FUNCTION_BLOCK FB_FeedForward
VAR_INPUT
	fXDotRef 	: LREAL; // Motion Referance
	fQMaxUp 	: LREAL; // Needs to be positive (22)
	fQMaxDown 	: LREAL; // Needs to be positive (15)
	fDeadUp		: LREAL; // Needs to be positive (0.155)
	fDeadDown 	: LREAL; // Needs to be positive (0.18)
	fPs 		: LREAL;
	fPa			: LREAL;
	fPb			: LREAL;
	fKFF 		: LREAL; // Coefficient of FeedForward
END_VAR
VAR_OUTPUT
	fUFF : LREAL;
END_VAR
VAR
	fUTemp : LREAL;
	fUMax : LREAL := 0.9;
	fQRef : LREAL;
	fAp : LREAL := 33.1 / 10000.0;
	fAa : LREAL := 23.56 / 10000.0;
	
	fK02Up : LREAL := 0.78; //0.78;
	fK04Up : LREAL := 2.29; //2.3;
	fK06Up : LREAL := 3.42;// 3.27;
	fK07Up : LREAL := 4.59; //4.54;
	fK08Up : LREAL := 5.09; //4.94;
	fK1Up : LREAL := 5.71; //5.68;
	
	fK02Down : LREAL := -0.75; //-0.75; 
	fK04Down : LREAL := -2.17; //-2.21; //-1.37;
	fK06Down : LREAL := -3.39; //-3.45; 
	fK07Down : LREAL := -3.99; //-3.96; //-2.45;
	fK08Down : LREAL := -4.55; //-4.61; 
	fK1Down : LREAL := -4.84; //-4.67; //-2.88;
	
	fDeltaP : LREAL;
	fKRef : LREAL; 
	
END_VAR



IF fXDotRef >= 0.0 THEN // Upwards
	
	fQRef := fAp * fXDotRef * 60000;
	fDeltaP := fPs - fPa;
	IF fDeltaP < 100 THEN
		fDeltaP := 100;
	ELSE
		fDeltaP := fDeltaP;
	END_IF
	fKRef := fQRef / SQRT(fDeltaP);
	
	IF fKRef < 0.0 THEN
		fUTemp := 0.0;
	ELSIF fKRef < fK02Up THEN
		fUTemp := -fKRef/fK02Up * (0.2 - fDeadUp);
	ELSIF fKRef < fK04Up THEN
		fUTemp := -(0.2 - fDeadUp) -(fKRef - fK02Up) / (fK04Up - fK02Up) * (0.4-fDeadUp-0.2);
	ELSIF fKRef < fK06Up THEN
		fUTemp := -(0.4 - fDeadUp - 0.2) - (0.2 - fDeadUp) - (fKRef - fK04Up) / (fK06Up - fK04Up) * (0.6-fDeadUp-0.4);
	ELSIF fKRef < fK07Up THEN
		fUTemp := -(0.6 - fDeadUp - 0.4) - (0.4 - fDeadUp - 0.2) - (0.2 - fDeadUp) - (fKRef - fK06Up) / (fK07Up - fK06Up) * (0.7 - fDeadUp - 0.6);
	ELSIF fKRef < fK08Up THEN
		fUTemp := -(0.7 - fDeadUp - 0.6) - (0.6 - fDeadUp - 0.4) - (0.4 - fDeadUp - 0.2 ) - (0.2 - fDeadUp) - (fKRef - fK07Up) / (fK08Up - fK07Up) * (0.8-fDeadUp-0.7);
	ELSIF fKRef < fK1Up THEN
		fUTemp := -(0.8 - fDeadUp - 0.7) - (0.7 - fDeadUp - 0.6) - (0.6 - fDeadUp - 0.4) - (0.4 - fDeadUp - 0.2 ) - (0.2 - fDeadUp) - (fKRef - fK08Up) / (fK1Up - fK08Up) * (1.0-fDeadUp-0.8);
	ELSE
		fUTemp := -(1 - fDeadUp);
	END_IF
	
//	fUTemp := -((fQRef/fQMaxUp) * (fUMax-fDeadUp));

ELSIF fXDotRef < 0.0 THEN // Downwards
	
	fQRef := fAa * fXDotRef * 60000;
	fDeltaP := fPs - fPb;
	IF fDeltaP < 100 THEN
		fDeltaP := 100;
	ELSE
		fDeltaP := fDeltaP;
	END_IF
	fKRef := fQRef / SQRT(fDeltaP);
	
	IF fKRef > 0.0 THEN
		fUTemp := 0.0;
	ELSIF fKRef > fK02Down THEN
		fUTemp := fKRef/fK02Down * (0.2-fDeadDown);
	ELSIF fKRef > fK04Down THEN
		fUTemp := (0.2 - fDeadDown) + (fKRef - fK02Down) / (fK04Down - fK02Down) * (0.4 - fDeadDown - 0.2);
	ELSIF fKRef > fK06Down THEN
		fUTemp := (0.2 - fDeadDown) + (0.4 - fDeadDown) + (fKRef - fK04Down) / (fK06Down - fK04Down) * (0.6 - fDeadDown - 0.4);
	ELSIF fKRef > fK07Down THEN
		fUTemp := (0.2 - fDeadDown) + (0.4 - fDeadDown) + (0.6 - fDeadDown) + (fKRef - fK06Down) / (fK07Down - fK06Down) * (0.7 - fDeadDown - 0.6);
	ELSIF fKRef > fK08Down THEN
		fUTemp := (0.2 - fDeadDown) + (0.4 - fDeadDown) + (0.6 - fDeadDown) + (0.7 - fDeadDown) + (fKRef - fK07Down) / (fK08Down - fK07Down) * (0.8 - fDeadDown - 0.7);
	ELSIF fKRef > fK1Down THEN
		fUTemp := (0.2 - fDeadDown) + (0.4 - fDeadDown) + (0.6 - fDeadDown) + (0.7 - fDeadDown) + (0.8 - fDeadDown) + (fKRef - fK08Down) / (fK1Down - fK08Down) * (1.0 - fDeadDown - 0.8);
	ELSE
		fUTemp := (1.0 - fDeadDown);
	END_IF
	
//	fUTemp := -((fQRef/fQMaxDown) * (fUMax-fDeadDown)); // FDeadDown needs to be positive
	

END_IF

fUFF := fUTemp * fKFF; // Tomec

END_FUNCTION_BLOCK

(* stored: Version 1.1.0.1, ProductVersion 3.1.4026.11
   POU FB_FeedForward: Id {c7c6c1c3-721c-4ea2-9006-d66030d86044}, SpecialFunc None *)
